(* PLC project LibIT_DO, lamsystems-it.ru LibIT_DO 1 *)
(* stored: creationDateTime 2019-11-13T09:37:45, productRelease 0, modificationDateTime 2023-01-20T15:46:21, version 1 *)

FUNCTION_BLOCK DOMode
  VAR_INPUT
    Ex : BOOL := FALSE;  (* разрешение на выполнение *)
    DOn : BYTE := 0;  (* номер выхода *)
    M : BYTE := 0;  (* режим работы *)
  END_VAR
  VAR_OUTPUT
    Ok : BYTE := 0;  (* код результата исполнения блока *)
  END_VAR

            {extern void App_DOMode(DOMODE*);App_DOMode(data__);}

          
END_FUNCTION_BLOCK

(* Текущий режим и состояние выхода DO *)
FUNCTION_BLOCK DOStatus
  VAR_INPUT
    DOn : BYTE := 0;  (* номер выхода *)
  END_VAR
  VAR_OUTPUT
    Om : BYTE := 0;  (* режим работы (установленный) *)
    Oepwm : BOOL := 0;  (* разрешение работы ШИМ (установленное) *)
    Otpwm : DWORD := 0;  (* период ШИМ (мс) *)
    Odpwm : REAL := 0.0;  (* коэффициент заполнения ШИМ (%) *)
    Oesf : BOOL := 0;  (* разрешение безопасного выхода (установленное) *)
    Ovsf : BOOL := 0;  (* значение безопасного выхода (установленное) *)
    Ok : BYTE := 0;  (* код результата исполнения блока *)
  END_VAR

            {extern void App_DOStatus(DOSTATUS*);App_DOStatus(data__);}

          
END_FUNCTION_BLOCK

FUNCTION_BLOCK DOVal
  VAR_INPUT
    Ex : BOOL := FALSE;  (* разрешение на выполнение *)
    DOn : BYTE := 0;  (* номер выхода *)
    V : BOOL := FALSE;  (* значение *)
  END_VAR
  VAR_OUTPUT
    Ov : BOOL := FALSE;  (* значение (установленное) *)
    Ok : BYTE := 0;  (* код результата исполнения блока *)
  END_VAR

            {extern void App_DOVal(DOVAL*);App_DOVal(data__);}

          
END_FUNCTION_BLOCK

(* Установка значения быстрого дискретного выхода *)
FUNCTION_BLOCK DOFast
  VAR_INPUT
    Ex : BOOL := FALSE;  (* разрешение на выполнение *)
    DOn : BYTE := 0;  (* номер выхода *)
    V : BOOL := FALSE;  (* значение *)
  END_VAR
  VAR_OUTPUT
    Ov : BOOL := FALSE;  (* значение (установленное) *)
  END_VAR
  VAR
    LastVal : BOOL := FALSE;  (* значение (установленное) *)
  END_VAR
  VAR_OUTPUT
    Ok : BYTE := 0;  (* код результата исполнения блока *)
  END_VAR

            {extern void App_DOFast(DOFAST*);App_DOFast(data__);}

          
END_FUNCTION_BLOCK

FUNCTION_BLOCK DOPwm
  VAR_INPUT
    Ex : BOOL := FALSE;  (* разрешение на выполнение *)
    EnPWM : BOOL := FALSE;  (* рашрешение работы ШИМ *)
    DOn : BYTE := 0;  (* номер выхода *)
    Tm : DWORD := 0;  (* период ШИМ (мс) *)
    Du : REAL := 0.0;  (* коэффициент заполнения ШИМ (%) *)
  END_VAR
  VAR_OUTPUT
    Ok : BYTE := 0;  (* код результата исполнения блока *)
  END_VAR

            {extern void App_DOPwm(DOPWM*);App_DOPwm(data__);}

          
END_FUNCTION_BLOCK

(* Установка значения безопасное состояния дискретного выхода *)
FUNCTION_BLOCK DOSafe
  VAR_INPUT
    Ex : BOOL := FALSE;  (* разрешение на выполнение *)
    EnSF : BOOL := FALSE;  (* разрешение безопасного выхода *)
    DOn : BYTE := 0;  (* номер выхода *)
    V : BOOL := FALSE;  (* значение безопасного выхода *)
  END_VAR
  VAR_OUTPUT
    Ok : BYTE := 0;  (* код результата исполнения блока *)
  END_VAR

            {extern void App_DOSafe(DOSAFE*);App_DOSafe(data__);}

          
END_FUNCTION_BLOCK
